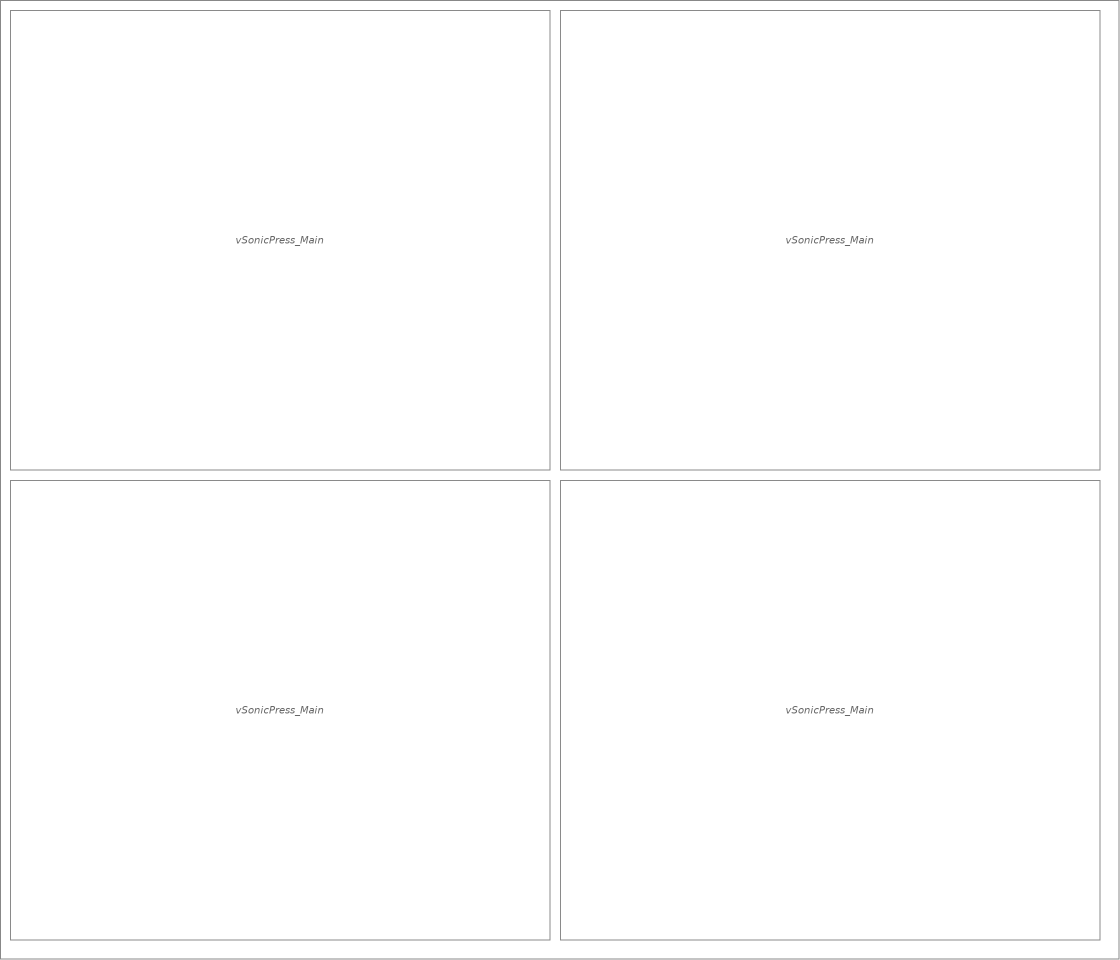
VISUALIZATION vS01_04  // 1120x960
    Frame (10,10 540x460)
        shows vSonicPress_Main(fbMachine := MAIN.fbS01_BearingPress, fbPIM := MAIN.fbS01_Station, stTestParams := stS01_TestParams)
    Frame (10,480 540x460)
        shows vSonicPress_Main(fbMachine := MAIN.fbS03_BearingPress, fbPIM := MAIN.fbS03_Station, stTestParams := stS03_TestParams)
    Frame (560,480 540x460)
        shows vSonicPress_Main(fbMachine := MAIN.fbS04_BearingPress, fbPIM := MAIN.fbS04_Station, stTestParams := stS04_TestParams)
    Frame (560,10 540x460)
        shows vSonicPress_Main(fbMachine := MAIN.fbS02_BearingPress, fbPIM := MAIN.fbS02_Station, stTestParams := stS02_TestParams)
END_VISUALIZATION

(* stored: Version 1.1.0.1, ProductVersion 3.1.4024.12
   Visu vS01_04: Id {ce78ed70-73de-42ed-bce3-06c0a45ba515} *)
